(* Logix 5000 project; controller Final vendor 1 type 14 code 242 rev 32.11; software revision 32.00; part 2 of 2 *)
(* tags used below, declared in another part *)
   B_Pres1 : SensorType;   // Holds all values related to Brakes Pressure Sensor #1
   B_Pres2 : SensorType;   // Holds all values related to Brakes Pressure Sensor #2
   B_Pres3 : SensorType;   // Holds all values related to Brakes Pressure Sensor #3
   B_Pres4 : SensorType;   // Holds all values related to Brakes Pressure Sensor #4
   B_Pres5 : SensorType;   // Holds all values related to Brakes Pressure Sensor #5
   B_Pres6 : SensorType;   // Holds all values related to Brakes Pressure Sensor #6
   B_Pres7 : SensorType;   // Holds all values related to Brakes Pressure Sensor #7
   B_Pres8 : SensorType;   // Holds all values related to Brakes Pressure Sensor #8
   B_Pres9 : SensorType;   // Holds all values related to Brakes Pressure Sensor #9
   B_Tem0 : SensorType;   // Holds all values related to Brakes Temperature Sensor #0
   B_Tem1 : SensorType;   // Holds all values related to Brakes Temperature Sensor #1
   BATTERY_CHARGE : REAL;
   BATTERY_TEMP : REAL;
   BATTERY_VOLTAGE : REAL;
   BatteryA : REAL;
   BatteryB : REAL;
   BatteryC : REAL;
   bfr_SysSec : DINT;
   C_Las0 : SensorType;   // Holds all values related to Controls Laser Sensor #0
   C_Las1 : SensorType;   // Holds all values related to Controls Laser Sensor #1
   ConversionResistance : REAL;
   ConversionVoltage : REAL;
   count : DINT;
   Current_OoR : BOOL;
   InverseTemp : REAL;
   Limit1 : BOOL;
   Limit2 : BOOL;
   LogR : REAL;
   P_Pres0 : SensorType;   // Holds all values related to Pressure Pressure Sensor #0
   P_Pres1 : SensorType;   // Holds all values related to Pressure Pressure Sensor #1
   P_Pres2 : SensorType;   // Holds all values related to Pressure Pressure Sensor #2
   P_Pres3 : SensorType;
   P_Pres4 : SensorType;
   P_Tem1 : SensorType;   // Holds all values related to Pressure Temperature Sensor #1
   P_Tem2 : SensorType;
   P_Tem3 : SensorType;
   P_Tem4 : SensorType;
   S_B_Pres0 : SensorType;
   S_B_Pres1 : SensorType;
   S_B_Pres2 : SensorType;
   S_B_Pres3 : SensorType;
   S_B_Pres4 : SensorType;
   S_B_Pres5 : SensorType;
   S_B_Pres6 : SensorType;
   S_B_Pres7 : SensorType;
   S_B_Pres8 : SensorType;
   S_B_Pres9 : SensorType;
   S_B_Tem0 : SensorType;
   S_B_Tem1 : SensorType;
   S_BAT_FLAG : BOOL;
   S_BatteryC : DINT;
   S_BatteryT : REAL;
   S_BatteryV : REAL;
   S_BRAKE_FLAG : BOOL;
   S_Brake_Sub1 : DINT;
   S_Brake_Sub2 : DINT;
   S_COMMAND : DINT;
   S_COMN_FLAG : BOOL;
   S_COMN_STATE : BOOL;
   S_P_Pres1 : SensorType;
   S_P_Pres2 : SensorType;
   S_P_Pres3 : SensorType;
   S_P_Pres4 : SensorType;
   S_P_Tem1 : SensorType;
   S_P_Tem2 : SensorType;
   S_P_Tem3 : SensorType;
   S_P_Tem4 : SensorType;
   S_PROP_FLAG : BOOL;
   S_PROP_STATE : BOOL;
   S_STATE : DINT;
   S_Switch : AB:5000_DO4:O:0;
   S_SysFail : BOOL;
   sts_SysSec : DINT;
   Temperature_OoR : BOOL;
   tmr_HB : TIMER;   // TIMER Heartbeat
   Voltage_OoR : BOOL;
(* MainProgram, continued *)

ROUTINE Update_B_Pres1   (* structured text *)
   case B_Pres1.Count of
   	0: B_Pres1.PreviousValue0 := B_Pres1.CurrentValue;
   	1: B_Pres1.PreviousValue1 := B_Pres1.CurrentValue;
   	2: B_Pres1.PreviousValue2 := B_Pres1.CurrentValue;
   	3: B_Pres1.PreviousValue3 := B_Pres1.CurrentValue;
   	4: B_Pres1.PreviousValue4 := B_Pres1.CurrentValue;
   	5: B_Pres1.PreviousValue5 := B_Pres1.CurrentValue;
   	6: B_Pres1.PreviousValue6 := B_Pres1.CurrentValue;
   	7: B_Pres1.PreviousValue7 := B_Pres1.CurrentValue;
   	8: B_Pres1.PreviousValue8 := B_Pres1.CurrentValue;
   	9: B_Pres1.PreviousValue9 := B_Pres1.CurrentValue;
   end_case;
   B_Pres1.Count := B_Pres1.Count + 1;
   if B_Pres1.Count = 10 then
   	B_Pres1.Count := 0;
   	B_Pres1.MeanStart := 1;
   end_if;
   B_Pres1.CurrentValue := Local:1:I.Ch01.Data;
   if B_Pres1.MeanStart then
   	B_Pres1.Mean10 := (B_Pres1.PreviousValue0 + B_Pres1.PreviousValue1 + B_Pres1.PreviousValue2 + B_Pres1.PreviousValue3 + B_Pres1.PreviousValue4 + B_Pres1.PreviousValue5 + B_Pres1.PreviousValue6 + B_Pres1.PreviousValue7 + B_Pres1.PreviousValue8 + B_Pres1.PreviousValue9)/10;
   	B_Pres1.StanDev := SQRT(( (B_Pres1.PreviousValue0 - B_Pres1.Mean10)**2 + (B_Pres1.PreviousValue1 - B_Pres1.Mean10)**2 + (B_Pres1.PreviousValue2 - B_Pres1.Mean10)**2 + (B_Pres1.PreviousValue3 - B_Pres1.Mean10)**2 + (B_Pres1.PreviousValue4 - B_Pres1.Mean10)**2 + (B_Pres1.PreviousValue5 - B_Pres1.Mean10)**2 + (B_Pres1.PreviousValue6 - B_Pres1.Mean10)**2 + (B_Pres1.PreviousValue7 - B_Pres1.Mean10)**2 + (B_Pres1.PreviousValue8 - B_Pres1.Mean10)**2 + (B_Pres1.PreviousValue9 - B_Pres1.Mean10)**2)/10);
   end_if;
END_ROUTINE

ROUTINE Update_B_Pres2   (* structured text *)
   case B_Pres2.Count of
   	0: B_Pres2.PreviousValue0 := B_Pres2.CurrentValue;
   	1: B_Pres2.PreviousValue1 := B_Pres2.CurrentValue;
   	2: B_Pres2.PreviousValue2 := B_Pres2.CurrentValue;
   	3: B_Pres2.PreviousValue3 := B_Pres2.CurrentValue;
   	4: B_Pres2.PreviousValue4 := B_Pres2.CurrentValue;
   	5: B_Pres2.PreviousValue5 := B_Pres2.CurrentValue;
   	6: B_Pres2.PreviousValue6 := B_Pres2.CurrentValue;
   	7: B_Pres2.PreviousValue7 := B_Pres2.CurrentValue;
   	8: B_Pres2.PreviousValue8 := B_Pres2.CurrentValue;
   	9: B_Pres2.PreviousValue9 := B_Pres2.CurrentValue;
   end_case;
   B_Pres2.Count := B_Pres2.Count + 1;
   if B_Pres2.Count = 10 then
   	B_Pres2.Count := 0;
   	B_Pres2.MeanStart := 1;
   end_if;
   B_Pres2.CurrentValue := Local:1:I.Ch02.Data;
   if B_Pres2.MeanStart then
   	B_Pres2.Mean10 := (B_Pres2.PreviousValue0 + B_Pres2.PreviousValue1 + B_Pres2.PreviousValue2 + B_Pres2.PreviousValue3 + B_Pres2.PreviousValue4 + B_Pres2.PreviousValue5 + B_Pres2.PreviousValue6 + B_Pres2.PreviousValue7 + B_Pres2.PreviousValue8 + B_Pres2.PreviousValue9)/10;
   	B_Pres2.StanDev := SQRT(((B_Pres2.PreviousValue0 - B_Pres2.Mean10)**2 + (B_Pres2.PreviousValue1 - B_Pres2.Mean10)**2 + (B_Pres2.PreviousValue2 - B_Pres2.Mean10)**2 + (B_Pres2.PreviousValue3 - B_Pres2.Mean10)**2 + (B_Pres2.PreviousValue4 - B_Pres2.Mean10)**2 + (B_Pres2.PreviousValue5 - B_Pres2.Mean10)**2 + (B_Pres2.PreviousValue6 - B_Pres2.Mean10)**2 + (B_Pres2.PreviousValue7 - B_Pres2.Mean10)**2 + (B_Pres2.PreviousValue8 - B_Pres2.Mean10)**2 + (B_Pres2.PreviousValue9 - B_Pres2.Mean10)**2)/10);
   end_if;
END_ROUTINE

ROUTINE Update_B_Pres3   (* structured text *)
   case B_Pres3.Count of
   	0: B_Pres3.PreviousValue0 := B_Pres3.CurrentValue;
   	1: B_Pres3.PreviousValue1 := B_Pres3.CurrentValue;
   	2: B_Pres3.PreviousValue2 := B_Pres3.CurrentValue;
   	3: B_Pres3.PreviousValue3 := B_Pres3.CurrentValue;
   	4: B_Pres3.PreviousValue4 := B_Pres3.CurrentValue;
   	5: B_Pres3.PreviousValue5 := B_Pres3.CurrentValue;
   	6: B_Pres3.PreviousValue6 := B_Pres3.CurrentValue;
   	7: B_Pres3.PreviousValue7 := B_Pres3.CurrentValue;
   	8: B_Pres3.PreviousValue8 := B_Pres3.CurrentValue;
   	9: B_Pres3.PreviousValue9 := B_Pres3.CurrentValue;
   end_case;
   B_Pres3.Count := B_Pres3.Count + 1;
   if B_Pres3.Count = 10 then
   	B_Pres3.Count := 0;
   	B_Pres3.MeanStart := 1;
   end_if;
   B_Pres3.CurrentValue := Local:1:I.Ch03.Data;
   if B_Pres3.MeanStart then
   	B_Pres3.Mean10 := (B_Pres3.PreviousValue0 + B_Pres3.PreviousValue1 + B_Pres3.PreviousValue2 + B_Pres3.PreviousValue3 + B_Pres3.PreviousValue4 + B_Pres3.PreviousValue5 + B_Pres3.PreviousValue6 + B_Pres3.PreviousValue7 + B_Pres3.PreviousValue8 + B_Pres3.PreviousValue9)/10;
   	B_Pres3.StanDev := SQRT(((B_Pres3.PreviousValue0 - B_Pres3.Mean10)**2 + (B_Pres3.PreviousValue1 - B_Pres3.Mean10)**2 + (B_Pres3.PreviousValue2 - B_Pres3.Mean10)**2 + (B_Pres3.PreviousValue3 - B_Pres3.Mean10)**2 + (B_Pres3.PreviousValue4 - B_Pres3.Mean10)**2 + (B_Pres3.PreviousValue5 - B_Pres3.Mean10)**2 + (B_Pres3.PreviousValue6 - B_Pres3.Mean10)**2 + (B_Pres3.PreviousValue7 - B_Pres3.Mean10)**2 + (B_Pres3.PreviousValue8 - B_Pres3.Mean10)**2 + (B_Pres3.PreviousValue9 - B_Pres3.Mean10)**2)/10);
   end_if;
END_ROUTINE

ROUTINE Update_B_Pres4   (* structured text *)
   case B_Pres4.Count of
   	0: B_Pres4.PreviousValue0 := B_Pres4.CurrentValue;
   	1: B_Pres4.PreviousValue1 := B_Pres4.CurrentValue;
   	2: B_Pres4.PreviousValue2 := B_Pres4.CurrentValue;
   	3: B_Pres4.PreviousValue3 := B_Pres4.CurrentValue;
   	4: B_Pres4.PreviousValue4 := B_Pres4.CurrentValue;
   	5: B_Pres4.PreviousValue5 := B_Pres4.CurrentValue;
   	6: B_Pres4.PreviousValue6 := B_Pres4.CurrentValue;
   	7: B_Pres4.PreviousValue7 := B_Pres4.CurrentValue;
   	8: B_Pres4.PreviousValue8 := B_Pres4.CurrentValue;
   	9: B_Pres4.PreviousValue9 := B_Pres4.CurrentValue;
   end_case;
   B_Pres4.Count := B_Pres4.Count + 1;
   if B_Pres4.Count = 10 then
   	B_Pres4.Count := 0;
   	B_Pres4.MeanStart := 1;
   end_if;
   B_Pres4.CurrentValue := Local:1:I.Ch04.Data;
   if B_Pres4.MeanStart then
   	B_Pres4.Mean10 := (B_Pres4.PreviousValue0 + B_Pres4.PreviousValue1 + B_Pres4.PreviousValue2 + B_Pres4.PreviousValue3 + B_Pres4.PreviousValue4 + B_Pres4.PreviousValue5 + B_Pres4.PreviousValue6 + B_Pres4.PreviousValue7 + B_Pres4.PreviousValue8 + B_Pres4.PreviousValue9)/10;
   	B_Pres4.StanDev := SQRT(((B_Pres4.PreviousValue0 - B_Pres4.Mean10)**2 + (B_Pres4.PreviousValue1 - B_Pres4.Mean10)**2 + (B_Pres4.PreviousValue2 - B_Pres4.Mean10)**2 + (B_Pres4.PreviousValue3 - B_Pres4.Mean10)**2 + (B_Pres4.PreviousValue4 - B_Pres4.Mean10)**2 + (B_Pres4.PreviousValue5 - B_Pres4.Mean10)**2 + (B_Pres4.PreviousValue6 - B_Pres4.Mean10)**2 + (B_Pres4.PreviousValue7 - B_Pres4.Mean10)**2 + (B_Pres4.PreviousValue8 - B_Pres4.Mean10)**2 + (B_Pres4.PreviousValue9 - B_Pres4.Mean10)**2)/10);
   end_if;
END_ROUTINE

ROUTINE Update_B_Pres5   (* structured text *)
   case B_Pres5.Count of
   	0: B_Pres5.PreviousValue0 := B_Pres5.CurrentValue;
   	1: B_Pres5.PreviousValue1 := B_Pres5.CurrentValue;
   	2: B_Pres5.PreviousValue2 := B_Pres5.CurrentValue;
   	3: B_Pres5.PreviousValue3 := B_Pres5.CurrentValue;
   	4: B_Pres5.PreviousValue4 := B_Pres5.CurrentValue;
   	5: B_Pres5.PreviousValue5 := B_Pres5.CurrentValue;
   	6: B_Pres5.PreviousValue6 := B_Pres5.CurrentValue;
   	7: B_Pres5.PreviousValue7 := B_Pres5.CurrentValue;
   	8: B_Pres5.PreviousValue8 := B_Pres5.CurrentValue;
   	9: B_Pres5.PreviousValue9 := B_Pres5.CurrentValue;
   end_case;
   B_Pres5.Count := B_Pres5.Count + 1;
   if B_Pres5.Count = 10 then
   	B_Pres5.Count := 0;
   	B_Pres5.MeanStart := 1;
   end_if;
   B_Pres5.CurrentValue := Local:1:I.Ch05.Data;
   if B_Pres5.MeanStart then
   	B_Pres5.Mean10 := (B_Pres5.PreviousValue0 + B_Pres5.PreviousValue1 + B_Pres5.PreviousValue2 + B_Pres5.PreviousValue3 + B_Pres5.PreviousValue4 + B_Pres5.PreviousValue5 + B_Pres5.PreviousValue6 + B_Pres5.PreviousValue7 + B_Pres5.PreviousValue8 + B_Pres5.PreviousValue9)/10;
   	B_Pres5.StanDev := SQRT(((B_Pres5.PreviousValue0 - B_Pres5.Mean10)**2 + (B_Pres5.PreviousValue1 - B_Pres5.Mean10)**2 + (B_Pres5.PreviousValue2 - B_Pres5.Mean10)**2 + (B_Pres5.PreviousValue3 - B_Pres5.Mean10)**2 + (B_Pres5.PreviousValue4 - B_Pres5.Mean10)**2 + (B_Pres5.PreviousValue5 - B_Pres5.Mean10)**2 + (B_Pres5.PreviousValue6 - B_Pres5.Mean10)**2 + (B_Pres5.PreviousValue7 - B_Pres5.Mean10)**2 + (B_Pres5.PreviousValue8 - B_Pres5.Mean10)**2 + (B_Pres5.PreviousValue9 - B_Pres5.Mean10)**2)/10);
   end_if;
END_ROUTINE

ROUTINE Update_B_Pres6   (* structured text *)
   case B_Pres6.Count of
   	0: B_Pres6.PreviousValue0 := B_Pres6.CurrentValue;
   	1: B_Pres6.PreviousValue1 := B_Pres6.CurrentValue;
   	2: B_Pres6.PreviousValue2 := B_Pres6.CurrentValue;
   	3: B_Pres6.PreviousValue3 := B_Pres6.CurrentValue;
   	4: B_Pres6.PreviousValue4 := B_Pres6.CurrentValue;
   	5: B_Pres6.PreviousValue5 := B_Pres6.CurrentValue;
   	6: B_Pres6.PreviousValue6 := B_Pres6.CurrentValue;
   	7: B_Pres6.PreviousValue7 := B_Pres6.CurrentValue;
   	8: B_Pres6.PreviousValue8 := B_Pres6.CurrentValue;
   	9: B_Pres6.PreviousValue9 := B_Pres6.CurrentValue;
   end_case;
   B_Pres6.Count := B_Pres6.Count + 1;
   if B_Pres6.Count = 10 then
   	B_Pres6.Count := 0;
   	B_Pres6.MeanStart := 1;
   end_if;
   B_Pres6.CurrentValue := Local:1:I.Ch06.Data;
   if B_Pres6.MeanStart then
   	B_Pres6.Mean10 := (B_Pres6.PreviousValue0 + B_Pres6.PreviousValue1 + B_Pres6.PreviousValue2 + B_Pres6.PreviousValue3 + B_Pres6.PreviousValue4 + B_Pres6.PreviousValue5 + B_Pres6.PreviousValue6 + B_Pres6.PreviousValue7 + B_Pres6.PreviousValue8 + B_Pres6.PreviousValue9)/10;
   	B_Pres6.StanDev := SQRT(((B_Pres6.PreviousValue0 - B_Pres6.Mean10)**2 + (B_Pres6.PreviousValue1 - B_Pres6.Mean10)**2 + (B_Pres6.PreviousValue2 - B_Pres6.Mean10)**2 + (B_Pres6.PreviousValue3 - B_Pres6.Mean10)**2 + (B_Pres6.PreviousValue4 - B_Pres6.Mean10)**2 + (B_Pres6.PreviousValue5 - B_Pres6.Mean10)**2 + (B_Pres6.PreviousValue6 - B_Pres6.Mean10)**2 + (B_Pres6.PreviousValue7 - B_Pres6.Mean10)**2 + (B_Pres6.PreviousValue8 - B_Pres6.Mean10)**2 + (B_Pres6.PreviousValue9 - B_Pres6.Mean10)**2)/10);
   end_if;
END_ROUTINE

ROUTINE Update_B_Pres7   (* structured text *)
   case B_Pres7.Count of
   	0: B_Pres7.PreviousValue0 := B_Pres7.CurrentValue;
   	1: B_Pres7.PreviousValue1 := B_Pres7.CurrentValue;
   	2: B_Pres7.PreviousValue2 := B_Pres7.CurrentValue;
   	3: B_Pres7.PreviousValue3 := B_Pres7.CurrentValue;
   	4: B_Pres7.PreviousValue4 := B_Pres7.CurrentValue;
   	5: B_Pres7.PreviousValue5 := B_Pres7.CurrentValue;
   	6: B_Pres7.PreviousValue6 := B_Pres7.CurrentValue;
   	7: B_Pres7.PreviousValue7 := B_Pres7.CurrentValue;
   	8: B_Pres7.PreviousValue8 := B_Pres7.CurrentValue;
   	9: B_Pres7.PreviousValue9 := B_Pres7.CurrentValue;
   end_case;
   B_Pres7.Count := B_Pres7.Count + 1;
   if B_Pres7.Count = 10 then
   	B_Pres7.Count := 0;
   	B_Pres7.MeanStart := 1;
   end_if;
   B_Pres7.CurrentValue := Local:1:I.Ch07.Data;
   if B_Pres7.MeanStart then
   	B_Pres7.Mean10 := (B_Pres7.PreviousValue0 + B_Pres7.PreviousValue1 + B_Pres7.PreviousValue2 + B_Pres7.PreviousValue3 + B_Pres7.PreviousValue4 + B_Pres7.PreviousValue5 + B_Pres7.PreviousValue6 + B_Pres7.PreviousValue7 + B_Pres7.PreviousValue8 + B_Pres7.PreviousValue9)/10;
   	B_Pres7.StanDev := SQRT(((B_Pres7.PreviousValue0 - B_Pres7.Mean10)**2 + (B_Pres7.PreviousValue1 - B_Pres7.Mean10)**2 + (B_Pres7.PreviousValue2 - B_Pres7.Mean10)**2 + (B_Pres7.PreviousValue3 - B_Pres7.Mean10)**2 + (B_Pres7.PreviousValue4 - B_Pres7.Mean10)**2 + (B_Pres7.PreviousValue5 - B_Pres7.Mean10)**2 + (B_Pres7.PreviousValue6 - B_Pres7.Mean10)**2 + (B_Pres7.PreviousValue7 - B_Pres7.Mean10)**2 + (B_Pres7.PreviousValue8 - B_Pres7.Mean10)**2 + (B_Pres7.PreviousValue9 - B_Pres7.Mean10)**2)/10);
   end_if;
END_ROUTINE

ROUTINE Update_B_Pres8   (* structured text *)
   case B_Pres8.Count of
   	0: B_Pres8.PreviousValue0 := B_Pres8.CurrentValue;
   	1: B_Pres8.PreviousValue1 := B_Pres8.CurrentValue;
   	2: B_Pres8.PreviousValue2 := B_Pres8.CurrentValue;
   	3: B_Pres8.PreviousValue3 := B_Pres8.CurrentValue;
   	4: B_Pres8.PreviousValue4 := B_Pres8.CurrentValue;
   	5: B_Pres8.PreviousValue5 := B_Pres8.CurrentValue;
   	6: B_Pres8.PreviousValue6 := B_Pres8.CurrentValue;
   	7: B_Pres8.PreviousValue7 := B_Pres8.CurrentValue;
   	8: B_Pres8.PreviousValue8 := B_Pres8.CurrentValue;
   	9: B_Pres8.PreviousValue9 := B_Pres8.CurrentValue;
   end_case;
   B_Pres8.Count := B_Pres8.Count + 1;
   if B_Pres8.Count = 10 then
   	B_Pres8.Count := 0;
   	B_Pres8.MeanStart := 1;
   end_if;
   B_Pres8.CurrentValue := Local:2:I.Ch00.Data;
   if B_Pres8.MeanStart then
   	B_Pres8.Mean10 := (B_Pres8.PreviousValue0 + B_Pres8.PreviousValue1 + B_Pres8.PreviousValue2 + B_Pres8.PreviousValue3 + B_Pres8.PreviousValue4 + B_Pres8.PreviousValue5 + B_Pres8.PreviousValue6 + B_Pres8.PreviousValue7 + B_Pres8.PreviousValue8 + B_Pres8.PreviousValue9)/10;
   	B_Pres8.StanDev := SQRT(((B_Pres8.PreviousValue0 - B_Pres8.Mean10)**2 + (B_Pres8.PreviousValue1 - B_Pres8.Mean10)**2 + (B_Pres8.PreviousValue2 - B_Pres8.Mean10)**2 + (B_Pres8.PreviousValue3 - B_Pres8.Mean10)**2 + (B_Pres8.PreviousValue4 - B_Pres8.Mean10)**2 + (B_Pres8.PreviousValue5 - B_Pres8.Mean10)**2 + (B_Pres8.PreviousValue6 - B_Pres8.Mean10)**2 + (B_Pres8.PreviousValue7 - B_Pres8.Mean10)**2 + (B_Pres8.PreviousValue8 - B_Pres8.Mean10)**2 + (B_Pres8.PreviousValue9 - B_Pres8.Mean10)**2)/10);
   end_if;
END_ROUTINE

ROUTINE Update_B_Pres9   (* structured text *)
   case B_Pres9.Count of
   	0: B_Pres9.PreviousValue0 := B_Pres9.CurrentValue;
   	1: B_Pres9.PreviousValue1 := B_Pres9.CurrentValue;
   	2: B_Pres9.PreviousValue2 := B_Pres9.CurrentValue;
   	3: B_Pres9.PreviousValue3 := B_Pres9.CurrentValue;
   	4: B_Pres9.PreviousValue4 := B_Pres9.CurrentValue;
   	5: B_Pres9.PreviousValue5 := B_Pres9.CurrentValue;
   	6: B_Pres9.PreviousValue6 := B_Pres9.CurrentValue;
   	7: B_Pres9.PreviousValue7 := B_Pres9.CurrentValue;
   	8: B_Pres9.PreviousValue8 := B_Pres9.CurrentValue;
   	9: B_Pres9.PreviousValue9 := B_Pres9.CurrentValue;
   end_case;
   B_Pres9.Count := B_Pres9.Count + 1;
   if B_Pres9.Count = 10 then
   	B_Pres9.Count := 0;
   	B_Pres9.MeanStart := 1;
   end_if;
   B_Pres9.CurrentValue := Local:2:I.Ch01.Data;
   if B_Pres9.MeanStart then
   	B_Pres9.Mean10 := (B_Pres9.PreviousValue0 + B_Pres9.PreviousValue1 + B_Pres9.PreviousValue2 + B_Pres9.PreviousValue3 + B_Pres9.PreviousValue4 + B_Pres9.PreviousValue5 + B_Pres9.PreviousValue6 + B_Pres9.PreviousValue7 + B_Pres9.PreviousValue8 + B_Pres9.PreviousValue9)/10;
   	B_Pres9.StanDev := SQRT(((B_Pres9.PreviousValue0 - B_Pres9.Mean10)**2 + (B_Pres9.PreviousValue1 - B_Pres9.Mean10)**2 + (B_Pres9.PreviousValue2 - B_Pres9.Mean10)**2 + (B_Pres9.PreviousValue3 - B_Pres9.Mean10)**2 + (B_Pres9.PreviousValue4 - B_Pres9.Mean10)**2 + (B_Pres9.PreviousValue5 - B_Pres9.Mean10)**2 + (B_Pres9.PreviousValue6 - B_Pres9.Mean10)**2 + (B_Pres9.PreviousValue7 - B_Pres9.Mean10)**2 + (B_Pres9.PreviousValue8 - B_Pres9.Mean10)**2 + (B_Pres9.PreviousValue9 - B_Pres9.Mean10)**2)/10);
   end_if;
END_ROUTINE

ROUTINE Update_B_Tem0   (* structured text *)
   case B_Tem0.Count of
   	0: B_Tem0.PreviousValue0 := B_Tem0.CurrentValue;
   	1: B_Tem0.PreviousValue1 := B_Tem0.CurrentValue;
   	2: B_Tem0.PreviousValue2 := B_Tem0.CurrentValue;
   	3: B_Tem0.PreviousValue3 := B_Tem0.CurrentValue;
   	4: B_Tem0.PreviousValue4 := B_Tem0.CurrentValue;
   	5: B_Tem0.PreviousValue5 := B_Tem0.CurrentValue;
   	6: B_Tem0.PreviousValue6 := B_Tem0.CurrentValue;
   	7: B_Tem0.PreviousValue7 := B_Tem0.CurrentValue;
   	8: B_Tem0.PreviousValue8 := B_Tem0.CurrentValue;
   	9: B_Tem0.PreviousValue9 := B_Tem0.CurrentValue;
   end_case;
   B_Tem0.Count := B_Tem0.Count + 1;
   if B_Tem0.Count = 10 then
   	B_Tem0.Count := 0;
   	B_Tem0.MeanStart := 1;
   end_if;
   B_Tem0.CurrentValue := Local:2:I.Ch02.Data;
   if B_Tem0.MeanStart then
   	B_Tem0.Mean10 := (B_Tem0.PreviousValue0 + B_Tem0.PreviousValue1 + B_Tem0.PreviousValue2 + B_Tem0.PreviousValue3 + B_Tem0.PreviousValue4 + B_Tem0.PreviousValue5 + B_Tem0.PreviousValue6 + B_Tem0.PreviousValue7 + B_Tem0.PreviousValue8 + B_Tem0.PreviousValue9)/10;
   	B_Tem0.StanDev := SQRT(((B_Tem0.PreviousValue0 - B_Tem0.Mean10)**2 + (B_Tem0.PreviousValue1 - B_Tem0.Mean10)**2 + (B_Tem0.PreviousValue2 - B_Tem0.Mean10)**2 + (B_Tem0.PreviousValue3 - B_Tem0.Mean10)**2 + (B_Tem0.PreviousValue4 - B_Tem0.Mean10)**2 + (B_Tem0.PreviousValue5 - B_Tem0.Mean10)**2 + (B_Tem0.PreviousValue6 - B_Tem0.Mean10)**2 + (B_Tem0.PreviousValue7 - B_Tem0.Mean10)**2 + (B_Tem0.PreviousValue8 - B_Tem0.Mean10)**2 + (B_Tem0.PreviousValue9 - B_Tem0.Mean10)**2)/10);
   end_if;
END_ROUTINE

ROUTINE Update_B_Tem1   (* structured text *)
   case B_Tem1.Count of
   	0: B_Tem1.PreviousValue0 := B_Tem1.CurrentValue;
   	1: B_Tem1.PreviousValue1 := B_Tem1.CurrentValue;
   	2: B_Tem1.PreviousValue2 := B_Tem1.CurrentValue;
   	3: B_Tem1.PreviousValue3 := B_Tem1.CurrentValue;
   	4: B_Tem1.PreviousValue4 := B_Tem1.CurrentValue;
   	5: B_Tem1.PreviousValue5 := B_Tem1.CurrentValue;
   	6: B_Tem1.PreviousValue6 := B_Tem1.CurrentValue;
   	7: B_Tem1.PreviousValue7 := B_Tem1.CurrentValue;
   	8: B_Tem1.PreviousValue8 := B_Tem1.CurrentValue;
   	9: B_Tem1.PreviousValue9 := B_Tem1.CurrentValue;
   end_case;
   B_Tem1.Count := B_Tem1.Count + 1;
   if B_Tem1.Count = 10 then
   	B_Tem1.Count := 0;
   	B_Tem1.MeanStart := 1;
   end_if;
   B_Tem1.CurrentValue := Local:2:I.Ch03.Data;
   if B_Tem1.MeanStart then
   	B_Tem1.Mean10 := (B_Tem1.PreviousValue0 + B_Tem1.PreviousValue1 + B_Tem1.PreviousValue2 + B_Tem1.PreviousValue3 + B_Tem1.PreviousValue4 + B_Tem1.PreviousValue5 + B_Tem1.PreviousValue6 + B_Tem1.PreviousValue7 + B_Tem1.PreviousValue8 + B_Tem1.PreviousValue9)/10;
   	B_Tem1.StanDev := SQRT(((B_Tem1.PreviousValue0 - B_Tem1.Mean10)**2 + (B_Tem1.PreviousValue1 - B_Tem1.Mean10)**2 + (B_Tem1.PreviousValue2 - B_Tem1.Mean10)**2 + (B_Tem1.PreviousValue3 - B_Tem1.Mean10)**2 + (B_Tem1.PreviousValue4 - B_Tem1.Mean10)**2 + (B_Tem1.PreviousValue5 - B_Tem1.Mean10)**2 + (B_Tem1.PreviousValue6 - B_Tem1.Mean10)**2 + (B_Tem1.PreviousValue7 - B_Tem1.Mean10)**2 + (B_Tem1.PreviousValue8 - B_Tem1.Mean10)**2 + (B_Tem1.PreviousValue9 - B_Tem1.Mean10)**2)/10);
   end_if;
END_ROUTINE

ROUTINE Update_Battery_Amp   (* structured text *)
   
END_ROUTINE

ROUTINE Update_Battery_Temp   (* structured text *)
   ConversionVoltage := Local:2:I.Ch06.Data;
   ConversionResistance := 12650 * (5 - ConversionVoltage) / ConversionVoltage;
   BatteryA := 0.00112924;//-0.0005697945479763659;//25.633751435943907;//
   BatteryB := 0.000234108;//0.0005112936453520823;//-20.64469507056110;//
   BatteryC := 0.000000087755;//-0.0000008923754330128293;//-0.338811414517226;//
   LogR := LN(ConversionResistance);
   InverseTemp := BatteryA + BatteryB * LogR + BatteryC * (LogR ** 3);
   BATTERY_TEMP := 1 / InverseTemp ;//- 45;
END_ROUTINE

ROUTINE Update_Battery_Volt   (* structured text *)
   BATTERY_VOLTAGE := Local:2:I.Ch05.Data;
   BATTERY_CHARGE := (BATTERY_VOLTAGE - 23) * 100 / 6;
END_ROUTINE

ROUTINE Update_C_Las0   (* structured text *)
   case C_Las0.Count of
   	0: C_Las0.PreviousValue0 := C_Las0.CurrentValue;
   	1: C_Las0.PreviousValue1 := C_Las0.CurrentValue;
   	2: C_Las0.PreviousValue2 := C_Las0.CurrentValue;
   	3: C_Las0.PreviousValue3 := C_Las0.CurrentValue;
   	4: C_Las0.PreviousValue4 := C_Las0.CurrentValue;
   	5: C_Las0.PreviousValue5 := C_Las0.CurrentValue;
   	6: C_Las0.PreviousValue6 := C_Las0.CurrentValue;
   	7: C_Las0.PreviousValue7 := C_Las0.CurrentValue;
   	8: C_Las0.PreviousValue8 := C_Las0.CurrentValue;
   	9: C_Las0.PreviousValue9 := C_Las0.CurrentValue;
   end_case;
   C_Las0.Count := C_Las0.Count + 1;
   if C_Las0.Count = 10 then
   	C_Las0.Count := 0;
   	C_Las0.MeanStart := 1;
   end_if;
   C_Las0.CurrentValue := Local:7:I.Counter00.Count;
   if C_Las0.MeanStart then
   	C_Las0.Mean10 := (C_Las0.PreviousValue0 + C_Las0.PreviousValue1 + C_Las0.PreviousValue2 + C_Las0.PreviousValue3 + C_Las0.PreviousValue4 + C_Las0.PreviousValue5 + C_Las0.PreviousValue6 + C_Las0.PreviousValue7 + C_Las0.PreviousValue8 + C_Las0.PreviousValue9)/10;
   	C_Las0.StanDev := SQRT(((C_Las0.PreviousValue0 - C_Las0.Mean10)**2 + (C_Las0.PreviousValue1 - C_Las0.Mean10)**2 + (C_Las0.PreviousValue2 - C_Las0.Mean10)**2 + (C_Las0.PreviousValue3 - C_Las0.Mean10)**2 + (C_Las0.PreviousValue4 - C_Las0.Mean10)**2 + (C_Las0.PreviousValue5 - C_Las0.Mean10)**2 + (C_Las0.PreviousValue6 - C_Las0.Mean10)**2 + (C_Las0.PreviousValue7 - C_Las0.Mean10)**2 + (C_Las0.PreviousValue8 - C_Las0.Mean10)**2 + (C_Las0.PreviousValue9 - C_Las0.Mean10)**2)/10);
   end_if;
END_ROUTINE

ROUTINE Update_C_Las1   (* structured text *)
   case C_Las1.Count of
   	0: C_Las1.PreviousValue0 := C_Las1.CurrentValue;
   	1: C_Las1.PreviousValue1 := C_Las1.CurrentValue;
   	2: C_Las1.PreviousValue2 := C_Las1.CurrentValue;
   	3: C_Las1.PreviousValue3 := C_Las1.CurrentValue;
   	4: C_Las1.PreviousValue4 := C_Las1.CurrentValue;
   	5: C_Las1.PreviousValue5 := C_Las1.CurrentValue;
   	6: C_Las1.PreviousValue6 := C_Las1.CurrentValue;
   	7: C_Las1.PreviousValue7 := C_Las1.CurrentValue;
   	8: C_Las1.PreviousValue8 := C_Las1.CurrentValue;
   	9: C_Las1.PreviousValue9 := C_Las1.CurrentValue;
   end_case;
   C_Las1.Count := C_Las1.Count + 1;
   if C_Las1.Count = 10 then
   	C_Las1.Count := 0;
   	C_Las1.MeanStart := 1;
   end_if;
   C_Las1.CurrentValue := Local:7:I.Counter01.Count;
   if C_Las1.MeanStart then
   	C_Las1.Mean10 := (C_Las1.PreviousValue0 + C_Las1.PreviousValue1 + C_Las1.PreviousValue2 + C_Las1.PreviousValue3 + C_Las1.PreviousValue4 + C_Las1.PreviousValue5 + C_Las1.PreviousValue6 + C_Las1.PreviousValue7 + C_Las1.PreviousValue8 + C_Las1.PreviousValue9)/10;
   	C_Las1.StanDev := SQRT(((C_Las1.PreviousValue0 - C_Las1.Mean10)**2 + (C_Las1.PreviousValue1 - C_Las1.Mean10)**2 + (C_Las1.PreviousValue2 - C_Las1.Mean10)**2 + (C_Las1.PreviousValue3 - C_Las1.Mean10)**2 + (C_Las1.PreviousValue4 - C_Las1.Mean10)**2 + (C_Las1.PreviousValue5 - C_Las1.Mean10)**2 + (C_Las1.PreviousValue6 - C_Las1.Mean10)**2 + (C_Las1.PreviousValue7 - C_Las1.Mean10)**2 + (C_Las1.PreviousValue8 - C_Las1.Mean10)**2 + (C_Las1.PreviousValue9 - C_Las1.Mean10)**2)/10);
   end_if;
END_ROUTINE

ROUTINE Update_Limit1   (* structured text *)
   Limit1 := Local:6:I.Pt00.Data;
END_ROUTINE

ROUTINE Update_Limit2   (* structured text *)
   Limit2 := Local:6:I.Pt01.Data;
END_ROUTINE

ROUTINE Update_P_Pres0   (* structured text *)
   case P_Pres0.Count of
   	0: P_Pres0.PreviousValue0 := P_Pres0.CurrentValue;
   	1: P_Pres0.PreviousValue1 := P_Pres0.CurrentValue;
   	2: P_Pres0.PreviousValue2 := P_Pres0.CurrentValue;
   	3: P_Pres0.PreviousValue3 := P_Pres0.CurrentValue;
   	4: P_Pres0.PreviousValue4 := P_Pres0.CurrentValue;
   	5: P_Pres0.PreviousValue5 := P_Pres0.CurrentValue;
   	6: P_Pres0.PreviousValue6 := P_Pres0.CurrentValue;
   	7: P_Pres0.PreviousValue7 := P_Pres0.CurrentValue;
   	8: P_Pres0.PreviousValue8 := P_Pres0.CurrentValue;
   	9: P_Pres0.PreviousValue9 := P_Pres0.CurrentValue;
   end_case;
   P_Pres0.Count := P_Pres0.Count + 1;
   if P_Pres0.Count = 10 then
   	P_Pres0.Count := 0;
   	P_Pres0.MeanStart := 1;
   end_if;
   P_Pres0.CurrentValue := Local:2:I.Ch04.Data;
   if P_Pres0.MeanStart then
   	P_Pres0.Mean10 := (P_Pres0.PreviousValue0 + P_Pres0.PreviousValue1 + P_Pres0.PreviousValue2 + P_Pres0.PreviousValue3 + P_Pres0.PreviousValue4 + P_Pres0.PreviousValue5 + P_Pres0.PreviousValue6 + P_Pres0.PreviousValue7 + P_Pres0.PreviousValue8 + P_Pres0.PreviousValue9)/10;
   	P_Pres0.StanDev := SQRT(((P_Pres0.PreviousValue0 - P_Pres0.Mean10)**2 + (P_Pres0.PreviousValue1 - P_Pres0.Mean10)**2 + (P_Pres0.PreviousValue2 - P_Pres0.Mean10)**2 + (P_Pres0.PreviousValue3 - P_Pres0.Mean10)**2 + (P_Pres0.PreviousValue4 - P_Pres0.Mean10)**2 + (P_Pres0.PreviousValue5 - P_Pres0.Mean10)**2 + (P_Pres0.PreviousValue6 - P_Pres0.Mean10)**2 + (P_Pres0.PreviousValue7 - P_Pres0.Mean10)**2 + (P_Pres0.PreviousValue8 - P_Pres0.Mean10)**2 + (P_Pres0.PreviousValue9 - P_Pres0.Mean10)**2)/10);
   end_if;
END_ROUTINE

ROUTINE Update_P_Pres1   (* structured text *)
   case P_Pres1.Count of
   	0: P_Pres1.PreviousValue0 := P_Pres1.CurrentValue;
   	1: P_Pres1.PreviousValue1 := P_Pres1.CurrentValue;
   	2: P_Pres1.PreviousValue2 := P_Pres1.CurrentValue;
   	3: P_Pres1.PreviousValue3 := P_Pres1.CurrentValue;
   	4: P_Pres1.PreviousValue4 := P_Pres1.CurrentValue;
   	5: P_Pres1.PreviousValue5 := P_Pres1.CurrentValue;
   	6: P_Pres1.PreviousValue6 := P_Pres1.CurrentValue;
   	7: P_Pres1.PreviousValue7 := P_Pres1.CurrentValue;
   	8: P_Pres1.PreviousValue8 := P_Pres1.CurrentValue;
   	9: P_Pres1.PreviousValue9 := P_Pres1.CurrentValue;
   end_case;
   P_Pres1.Count := P_Pres1.Count + 1;
   if P_Pres1.Count = 10 then
   	P_Pres1.Count := 0;
   	P_Pres0.MeanStart := 1;
   end_if;
   P_Pres1.CurrentValue := Local:3:I.Ch00.Data;
   if P_Pres1.MeanStart then
   	P_Pres1.Mean10 := (P_Pres1.PreviousValue0 + P_Pres1.PreviousValue1 + P_Pres1.PreviousValue2 + P_Pres1.PreviousValue3 + P_Pres1.PreviousValue4 + P_Pres1.PreviousValue5 + P_Pres1.PreviousValue6 + P_Pres1.PreviousValue7 + P_Pres1.PreviousValue8 + P_Pres1.PreviousValue9)/10;
   	P_Pres1.StanDev := SQRT(((P_Pres1.PreviousValue0 - P_Pres1.Mean10)**2 + (P_Pres1.PreviousValue1 - P_Pres1.Mean10)**2 + (P_Pres1.PreviousValue2 - P_Pres1.Mean10)**2 + (P_Pres1.PreviousValue3 - P_Pres1.Mean10)**2 + (P_Pres1.PreviousValue4 - P_Pres1.Mean10)**2 + (P_Pres1.PreviousValue5 - P_Pres1.Mean10)**2 + (P_Pres1.PreviousValue6 - P_Pres1.Mean10)**2 + (P_Pres1.PreviousValue7 - P_Pres1.Mean10)**2 + (P_Pres1.PreviousValue8 - P_Pres1.Mean10)**2 + (P_Pres1.PreviousValue9 - P_Pres1.Mean10)**2)/10);
   end_if;
END_ROUTINE

ROUTINE Update_P_Pres2   (* structured text *)
   case P_Pres2.Count of
   	0: P_Pres2.PreviousValue0 := P_Pres2.CurrentValue;
   	1: P_Pres2.PreviousValue1 := P_Pres2.CurrentValue;
   	2: P_Pres2.PreviousValue2 := P_Pres2.CurrentValue;
   	3: P_Pres2.PreviousValue3 := P_Pres2.CurrentValue;
   	4: P_Pres2.PreviousValue4 := P_Pres2.CurrentValue;
   	5: P_Pres2.PreviousValue5 := P_Pres2.CurrentValue;
   	6: P_Pres2.PreviousValue6 := P_Pres2.CurrentValue;
   	7: P_Pres2.PreviousValue7 := P_Pres2.CurrentValue;
   	8: P_Pres2.PreviousValue8 := P_Pres2.CurrentValue;
   	9: P_Pres2.PreviousValue9 := P_Pres2.CurrentValue;
   end_case;
   P_Pres2.Count := P_Pres2.Count + 1;
   if P_Pres2.Count = 10 then
   	P_Pres2.Count := 0;
   	P_Pres2.MeanStart := 1;
   end_if;
   P_Pres2.CurrentValue := Local:3:I.Ch01.Data;
   if P_Pres2.MeanStart then
   	P_Pres2.Mean10 := (P_Pres2.PreviousValue0 + P_Pres2.PreviousValue1 + P_Pres2.PreviousValue2 + P_Pres2.PreviousValue3 + P_Pres2.PreviousValue4 + P_Pres2.PreviousValue5 + P_Pres2.PreviousValue6 + P_Pres2.PreviousValue7 + P_Pres2.PreviousValue8 + P_Pres2.PreviousValue9)/10;
   	P_Pres2.StanDev := SQRT(((P_Pres2.PreviousValue0 - P_Pres2.Mean10)**2 + (P_Pres2.PreviousValue1 - P_Pres2.Mean10)**2 + (P_Pres2.PreviousValue2 - P_Pres2.Mean10)**2 + (P_Pres2.PreviousValue3 - P_Pres2.Mean10)**2 + (P_Pres2.PreviousValue4 - P_Pres2.Mean10)**2 + (P_Pres2.PreviousValue5 - P_Pres2.Mean10)**2 + (P_Pres2.PreviousValue6 - P_Pres2.Mean10)**2 + (P_Pres2.PreviousValue7 - P_Pres2.Mean10)**2 + (P_Pres2.PreviousValue8 - P_Pres2.Mean10)**2 + (P_Pres2.PreviousValue9 - P_Pres2.Mean10)**2)/10);
   end_if;
END_ROUTINE

ROUTINE Update_P_Pres3   (* structured text *)
   case P_Pres3.Count of
   	0: P_Pres3.PreviousValue0 := P_Pres3.CurrentValue;
   	1: P_Pres3.PreviousValue1 := P_Pres3.CurrentValue;
   	2: P_Pres3.PreviousValue2 := P_Pres3.CurrentValue;
   	3: P_Pres3.PreviousValue3 := P_Pres3.CurrentValue;
   	4: P_Pres3.PreviousValue4 := P_Pres3.CurrentValue;
   	5: P_Pres3.PreviousValue5 := P_Pres3.CurrentValue;
   	6: P_Pres3.PreviousValue6 := P_Pres3.CurrentValue;
   	7: P_Pres3.PreviousValue7 := P_Pres3.CurrentValue;
   	8: P_Pres3.PreviousValue8 := P_Pres3.CurrentValue;
   	9: P_Pres3.PreviousValue9 := P_Pres3.CurrentValue;
   end_case;
   P_Pres3.Count := P_Pres3.Count + 1;
   if P_Pres3.Count = 10 then
   	P_Pres3.Count := 0;
   	P_Pres3.MeanStart := 1;
   end_if;
   P_Pres3.CurrentValue := Local:3:I.Ch02.Data;
   if P_Pres3.MeanStart then
   	P_Pres3.Mean10 := (P_Pres3.PreviousValue0 + P_Pres3.PreviousValue1 + P_Pres3.PreviousValue2 + P_Pres3.PreviousValue3 + P_Pres3.PreviousValue4 + P_Pres3.PreviousValue5 + P_Pres3.PreviousValue6 + P_Pres3.PreviousValue7 + P_Pres3.PreviousValue8 + P_Pres3.PreviousValue9)/10;
   	P_Pres3.StanDev := SQRT(((P_Pres3.PreviousValue0 - P_Pres3.Mean10)**2 + (P_Pres3.PreviousValue1 - P_Pres3.Mean10)**2 + (P_Pres3.PreviousValue2 - P_Pres3.Mean10)**2 + (P_Pres3.PreviousValue3 - P_Pres3.Mean10)**2 + (P_Pres3.PreviousValue4 - P_Pres3.Mean10)**2 + (P_Pres3.PreviousValue5 - P_Pres3.Mean10)**2 + (P_Pres3.PreviousValue6 - P_Pres3.Mean10)**2 + (P_Pres3.PreviousValue7 - P_Pres3.Mean10)**2 + (P_Pres3.PreviousValue8 - P_Pres3.Mean10)**2 + (P_Pres3.PreviousValue9 - P_Pres3.Mean10)**2)/10);
   end_if;
END_ROUTINE

ROUTINE Update_P_Pres4   (* structured text *)
   case P_Pres4.Count of
   	0: P_Pres4.PreviousValue0 := P_Pres4.CurrentValue;
   	1: P_Pres4.PreviousValue1 := P_Pres4.CurrentValue;
   	2: P_Pres4.PreviousValue2 := P_Pres4.CurrentValue;
   	3: P_Pres4.PreviousValue3 := P_Pres4.CurrentValue;
   	4: P_Pres4.PreviousValue4 := P_Pres4.CurrentValue;
   	5: P_Pres4.PreviousValue5 := P_Pres4.CurrentValue;
   	6: P_Pres4.PreviousValue6 := P_Pres4.CurrentValue;
   	7: P_Pres4.PreviousValue7 := P_Pres4.CurrentValue;
   	8: P_Pres4.PreviousValue8 := P_Pres4.CurrentValue;
   	9: P_Pres4.PreviousValue9 := P_Pres4.CurrentValue;
   end_case;
   P_Pres4.Count := P_Pres4.Count + 1;
   if P_Pres4.Count = 10 then
   	P_Pres4.Count := 0;
   	P_Pres4.MeanStart := 1;
   end_if;
   P_Pres4.CurrentValue := Local:3:I.Ch03.Data;
   if P_Pres4.MeanStart then
   	P_Pres4.Mean10 := (P_Pres4.PreviousValue0 + P_Pres4.PreviousValue1 + P_Pres4.PreviousValue2 + P_Pres4.PreviousValue3 + P_Pres4.PreviousValue4 + P_Pres4.PreviousValue5 + P_Pres4.PreviousValue6 + P_Pres4.PreviousValue7 + P_Pres4.PreviousValue8 + P_Pres4.PreviousValue9)/10;
   	P_Pres4.StanDev := SQRT(((P_Pres4.PreviousValue0 - P_Pres4.Mean10)**2 + (P_Pres4.PreviousValue1 - P_Pres4.Mean10)**2 + (P_Pres4.PreviousValue2 - P_Pres4.Mean10)**2 + (P_Pres4.PreviousValue3 - P_Pres4.Mean10)**2 + (P_Pres4.PreviousValue4 - P_Pres4.Mean10)**2 + (P_Pres4.PreviousValue5 - P_Pres4.Mean10)**2 + (P_Pres4.PreviousValue6 - P_Pres4.Mean10)**2 + (P_Pres4.PreviousValue7 - P_Pres4.Mean10)**2 + (P_Pres4.PreviousValue8 - P_Pres4.Mean10)**2 + (P_Pres4.PreviousValue9 - P_Pres4.Mean10)**2)/10);
   end_if;
END_ROUTINE

ROUTINE Update_P_Tem1   (* structured text *)
   case P_Tem1.Count of
   	0: P_Tem1.PreviousValue0 := P_Tem1.CurrentValue;
   	1: P_Tem1.PreviousValue1 := P_Tem1.CurrentValue;
   	2: P_Tem1.PreviousValue2 := P_Tem1.CurrentValue;
   	3: P_Tem1.PreviousValue3 := P_Tem1.CurrentValue;
   	4: P_Tem1.PreviousValue4 := P_Tem1.CurrentValue;
   	5: P_Tem1.PreviousValue5 := P_Tem1.CurrentValue;
   	6: P_Tem1.PreviousValue6 := P_Tem1.CurrentValue;
   	7: P_Tem1.PreviousValue7 := P_Tem1.CurrentValue;
   	8: P_Tem1.PreviousValue8 := P_Tem1.CurrentValue;
   	9: P_Tem1.PreviousValue9 := P_Tem1.CurrentValue;
   end_case;
   P_Tem1.Count := P_Tem1.Count + 1;
   if P_Tem1.Count = 10 then
   	P_Tem1.Count := 0;
   	P_Tem1.MeanStart := 1;
   end_if;
   P_Tem1.CurrentValue := Local:3:I.Ch04.Data;
   if P_Tem1.MeanStart then
   	P_Tem1.Mean10 := (P_Tem1.PreviousValue0 + P_Tem1.PreviousValue1 + P_Tem1.PreviousValue2 + P_Tem1.PreviousValue3 + P_Tem1.PreviousValue4 + P_Tem1.PreviousValue5 + P_Tem1.PreviousValue6 + P_Tem1.PreviousValue7 + P_Tem1.PreviousValue8 + P_Tem1.PreviousValue9)/10;
   	P_Tem1.StanDev := SQRT(((P_Tem1.PreviousValue0 - P_Tem1.Mean10)**2 + (P_Tem1.PreviousValue1 - P_Tem1.Mean10)**2 + (P_Tem1.PreviousValue2 - P_Tem1.Mean10)**2 + (P_Tem1.PreviousValue3 - P_Tem1.Mean10)**2 + (P_Tem1.PreviousValue4 - P_Tem1.Mean10)**2 + (P_Tem1.PreviousValue5 - P_Tem1.Mean10)**2 + (P_Tem1.PreviousValue6 - P_Tem1.Mean10)**2 + (P_Tem1.PreviousValue7 - P_Tem1.Mean10)**2 + (P_Tem1.PreviousValue8 - P_Tem1.Mean10)**2 + (P_Tem1.PreviousValue9 - P_Tem1.Mean10)**2)/10);
   end_if;
END_ROUTINE

ROUTINE Update_P_Tem2   (* structured text *)
   case P_Tem2.Count of
   	0: P_Tem2.PreviousValue0 := P_Tem2.CurrentValue;
   	1: P_Tem2.PreviousValue1 := P_Tem2.CurrentValue;
   	2: P_Tem2.PreviousValue2 := P_Tem2.CurrentValue;
   	3: P_Tem2.PreviousValue3 := P_Tem2.CurrentValue;
   	4: P_Tem2.PreviousValue4 := P_Tem2.CurrentValue;
   	5: P_Tem2.PreviousValue5 := P_Tem2.CurrentValue;
   	6: P_Tem2.PreviousValue6 := P_Tem2.CurrentValue;
   	7: P_Tem2.PreviousValue7 := P_Tem2.CurrentValue;
   	8: P_Tem2.PreviousValue8 := P_Tem2.CurrentValue;
   	9: P_Tem2.PreviousValue9 := P_Tem2.CurrentValue;
   end_case;
   P_Tem2.Count := P_Tem2.Count + 1;
   if P_Tem2.Count = 10 then
   	P_Tem2.Count := 0;
   	P_Tem2.MeanStart := 1;
   end_if;
   P_Tem2.CurrentValue := Local:3:I.Ch05.Data;
   if P_Tem2.MeanStart then
   	P_Tem2.Mean10 := (P_Tem2.PreviousValue0 + P_Tem2.PreviousValue1 + P_Tem2.PreviousValue2 + P_Tem2.PreviousValue3 + P_Tem2.PreviousValue4 + P_Tem2.PreviousValue5 + P_Tem2.PreviousValue6 + P_Tem2.PreviousValue7 + P_Tem2.PreviousValue8 + P_Tem2.PreviousValue9)/10;
   	P_Tem2.StanDev := SQRT(((P_Tem2.PreviousValue0 - P_Tem2.Mean10)**2 + (P_Tem2.PreviousValue1 - P_Tem2.Mean10)**2 + (P_Tem2.PreviousValue2 - P_Tem2.Mean10)**2 + (P_Tem2.PreviousValue3 - P_Tem2.Mean10)**2 + (P_Tem2.PreviousValue4 - P_Tem2.Mean10)**2 + (P_Tem2.PreviousValue5 - P_Tem2.Mean10)**2 + (P_Tem2.PreviousValue6 - P_Tem2.Mean10)**2 + (P_Tem2.PreviousValue7 - P_Tem2.Mean10)**2 + (P_Tem2.PreviousValue8 - P_Tem2.Mean10)**2 + (P_Tem2.PreviousValue9 - P_Tem2.Mean10)**2)/10);
   end_if;
END_ROUTINE

ROUTINE Update_P_Tem3   (* structured text *)
   case P_Tem3.Count of
   	0: P_Tem3.PreviousValue0 := P_Tem3.CurrentValue;
   	1: P_Tem3.PreviousValue1 := P_Tem3.CurrentValue;
   	2: P_Tem3.PreviousValue2 := P_Tem3.CurrentValue;
   	3: P_Tem3.PreviousValue3 := P_Tem3.CurrentValue;
   	4: P_Tem3.PreviousValue4 := P_Tem3.CurrentValue;
   	5: P_Tem3.PreviousValue5 := P_Tem3.CurrentValue;
   	6: P_Tem3.PreviousValue6 := P_Tem3.CurrentValue;
   	7: P_Tem3.PreviousValue7 := P_Tem3.CurrentValue;
   	8: P_Tem3.PreviousValue8 := P_Tem3.CurrentValue;
   	9: P_Tem3.PreviousValue9 := P_Tem3.CurrentValue;
   end_case;
   P_Tem3.Count := P_Tem3.Count + 1;
   if P_Tem3.Count = 10 then
   	P_Tem3.Count := 0;
   	P_Tem3.MeanStart := 1;
   end_if;
   P_Tem3.CurrentValue := Local:3:I.Ch06.Data;
   if P_Tem3.MeanStart then
   	P_Tem3.Mean10 := (P_Tem3.PreviousValue0 + P_Tem3.PreviousValue1 + P_Tem3.PreviousValue2 + P_Tem3.PreviousValue3 + P_Tem3.PreviousValue4 + P_Tem3.PreviousValue5 + P_Tem3.PreviousValue6 + P_Tem3.PreviousValue7 + P_Tem3.PreviousValue8 + P_Tem3.PreviousValue9)/10;
   	P_Tem3.StanDev := SQRT(((P_Tem3.PreviousValue0 - P_Tem3.Mean10)**2 + (P_Tem3.PreviousValue1 - P_Tem3.Mean10)**2 + (P_Tem3.PreviousValue2 - P_Tem3.Mean10)**2 + (P_Tem3.PreviousValue3 - P_Tem3.Mean10)**2 + (P_Tem3.PreviousValue4 - P_Tem3.Mean10)**2 + (P_Tem3.PreviousValue5 - P_Tem3.Mean10)**2 + (P_Tem3.PreviousValue6 - P_Tem3.Mean10)**2 + (P_Tem3.PreviousValue7 - P_Tem3.Mean10)**2 + (P_Tem3.PreviousValue8 - P_Tem3.Mean10)**2 + (P_Tem3.PreviousValue9 - P_Tem3.Mean10)**2)/10);
   end_if;
END_ROUTINE

ROUTINE Update_P_Tem4   (* structured text *)
   case P_Tem4.Count of
   	0: P_Tem4.PreviousValue0 := P_Tem4.CurrentValue;
   	1: P_Tem4.PreviousValue1 := P_Tem4.CurrentValue;
   	2: P_Tem4.PreviousValue2 := P_Tem4.CurrentValue;
   	3: P_Tem4.PreviousValue3 := P_Tem4.CurrentValue;
   	4: P_Tem4.PreviousValue4 := P_Tem4.CurrentValue;
   	5: P_Tem4.PreviousValue5 := P_Tem4.CurrentValue;
   	6: P_Tem4.PreviousValue6 := P_Tem4.CurrentValue;
   	7: P_Tem4.PreviousValue7 := P_Tem4.CurrentValue;
   	8: P_Tem4.PreviousValue8 := P_Tem4.CurrentValue;
   	9: P_Tem4.PreviousValue9 := P_Tem4.CurrentValue;
   end_case;
   P_Tem4.Count := P_Tem4.Count + 1;
   if P_Tem4.Count = 10 then
   	P_Tem4.Count := 0;
   	P_Tem4.MeanStart := 1;
   end_if;
   P_Tem4.CurrentValue := Local:3:I.Ch07.Data;
   if P_Tem4.MeanStart then
   	P_Tem4.Mean10 := (P_Tem4.PreviousValue0 + P_Tem4.PreviousValue1 + P_Tem4.PreviousValue2 + P_Tem4.PreviousValue3 + P_Tem4.PreviousValue4 + P_Tem4.PreviousValue5 + P_Tem4.PreviousValue6 + P_Tem4.PreviousValue7 + P_Tem4.PreviousValue8 + P_Tem4.PreviousValue9)/10;
   	P_Tem4.StanDev := SQRT(((P_Tem4.PreviousValue0 - P_Tem4.Mean10)**2 + (P_Tem4.PreviousValue1 - P_Tem4.Mean10)**2 + (P_Tem4.PreviousValue2 - P_Tem4.Mean10)**2 + (P_Tem4.PreviousValue3 - P_Tem4.Mean10)**2 + (P_Tem4.PreviousValue4 - P_Tem4.Mean10)**2 + (P_Tem4.PreviousValue5 - P_Tem4.Mean10)**2 + (P_Tem4.PreviousValue6 - P_Tem4.Mean10)**2 + (P_Tem4.PreviousValue7 - P_Tem4.Mean10)**2 + (P_Tem4.PreviousValue8 - P_Tem4.Mean10)**2 + (P_Tem4.PreviousValue9 - P_Tem4.Mean10)**2)/10);
   end_if;
END_ROUTINE
END_PROGRAM

PROGRAM SafetyProgram   (* main routine MainRoutine, safety *)
VAR
   B_Stage1 : BOOL;
   B_Stage2 : BOOL;
END_VAR

ROUTINE Eval_Bat   (* ladder *)
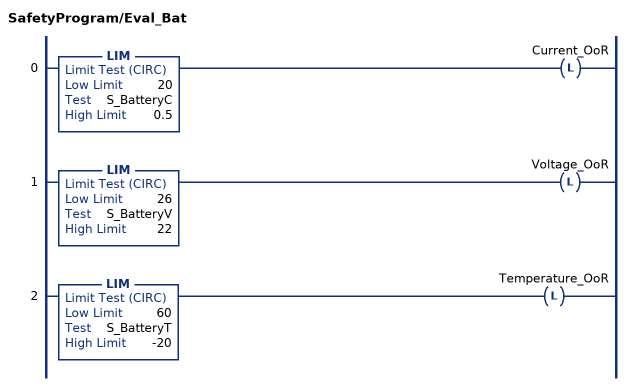
   0: LIM(20,S_BatteryC,0.5)OTL(Current_OoR);
   1: LIM(26,S_BatteryV,22)OTL(Voltage_OoR);
   2: LIM(60,S_BatteryT,-20)OTL(Temperature_OoR);
END_ROUTINE

ROUTINE Eval_Brake   (* ladder *)
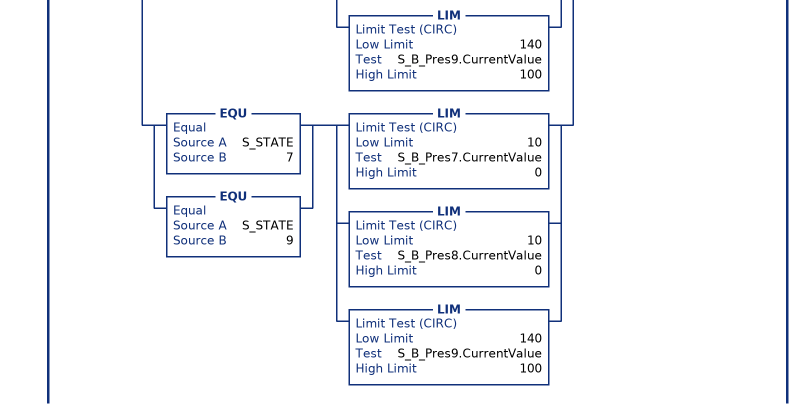
   0: [OTL(B_Stage1) [[LIM(105,S_B_Pres0.CurrentValue,95) ,LIM(105,S_B_Pres1.CurrentValue,95) ,LIM(30,S_B_Tem0.CurrentValue,20) ] ,[LIM(1,S_STATE,5) ,EQU(S_STATE,8) ] [LIM(16,S_B_Pres2.CurrentValue,12) ,LIM(16,S_B_Pres3.CurrentValue,12) ,LIM(170,S_B_Pres4.CurrentValue,150) ] ,[EQU(S_STATE,6) ,EQU(S_STATE,10) ] [LIM(105,S_B_Pres2.CurrentValue,95) ,LIM(105,S_B_Pres3.CurrentValue,95) ,LIM(140,S_B_Pres4.CurrentValue,100) ] ,[EQU(S_STATE,7) ,EQU(S_STATE,9) ] [LIM(10,S_B_Pres2.CurrentValue,0) ,LIM(10,S_B_Pres3.CurrentValue,0) ,LIM(140,S_B_Pres4.CurrentValue,100) ] ] MOV(1,S_Brake_Sub1) ,OTL(B_Stage2) [[LIM(105,S_B_Pres5.CurrentValue,95) ,LIM(105,S_B_Pres6.CurrentValue,95) ,LIM(30,S_B_Tem1.CurrentValue,20) ] ,[LIM(1,S_STATE,5) ,EQU(S_STATE,8) ] [LIM(16,S_B_Pres7.CurrentValue,12) ,LIM(16,S_B_Pres8.CurrentValue,12) ,LIM(170,S_B_Pres9.CurrentValue,150) ] ,[EQU(S_STATE,6) ,EQU(S_STATE,10) ] [LIM(105,S_B_Pres7.CurrentValue,95) ,LIM(105,S_B_Pres8.CurrentValue,95) ,LIM(140,S_B_Pres9.CurrentValue,100) ] ,[EQU(S_STATE,7) ,EQU(S_STATE,9) ] [LIM(10,S_B_Pres7.CurrentValue,0) ,LIM(10,S_B_Pres8.CurrentValue,0) ,LIM(140,S_B_Pres9.CurrentValue,100) ] ] MOV(1,S_Brake_Sub2) ];
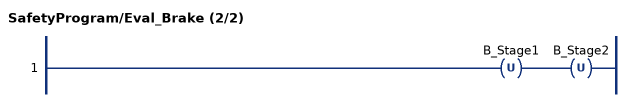
   1: OTU(B_Stage1)OTU(B_Stage2);
END_ROUTINE

ROUTINE Eval_Comm   (* ladder *)
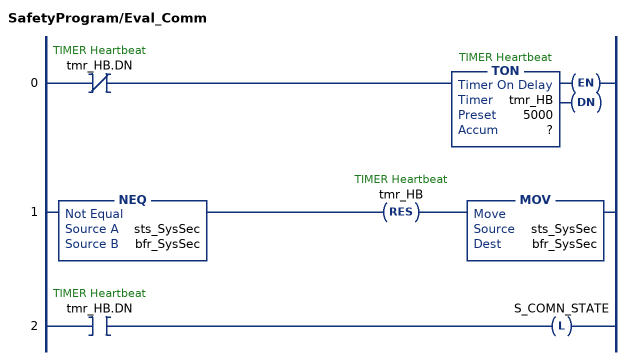
   0: XIO(tmr_HB.DN)TON(tmr_HB,?,?);
   1: NEQ(sts_SysSec,bfr_SysSec)RES(tmr_HB)MOV(sts_SysSec,bfr_SysSec);
   2: XIC(tmr_HB.DN)OTL(S_COMN_STATE);
END_ROUTINE

ROUTINE Eval_Prop   (* ladder *)
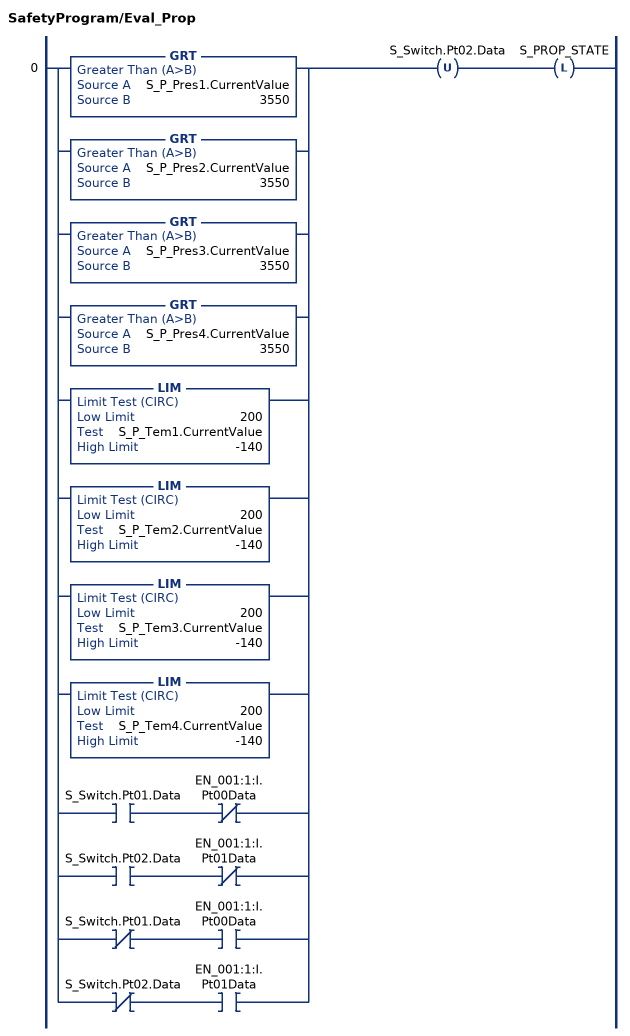
   0: [GRT(S_P_Pres1.CurrentValue,3550) ,GRT(S_P_Pres2.CurrentValue,3550) ,GRT(S_P_Pres3.CurrentValue,3550) ,GRT(S_P_Pres4.CurrentValue,3550) ,LIM(200,S_P_Tem1.CurrentValue,-140) ,LIM(200,S_P_Tem2.CurrentValue,-140) ,LIM(200,S_P_Tem3.CurrentValue,-140) ,LIM(200,S_P_Tem4.CurrentValue,-140) ,XIC(S_Switch.Pt01.Data) XIO(EN_001:1:I.Pt00Data) ,XIC(S_Switch.Pt02.Data) XIO(EN_001:1:I.Pt01Data) ,XIO(S_Switch.Pt01.Data) XIC(EN_001:1:I.Pt00Data) ,XIO(S_Switch.Pt02.Data) XIC(EN_001:1:I.Pt01Data) ]OTU(S_Switch.Pt02.Data)OTL(S_PROP_STATE);
END_ROUTINE

ROUTINE MainRoutine   (* ladder *)
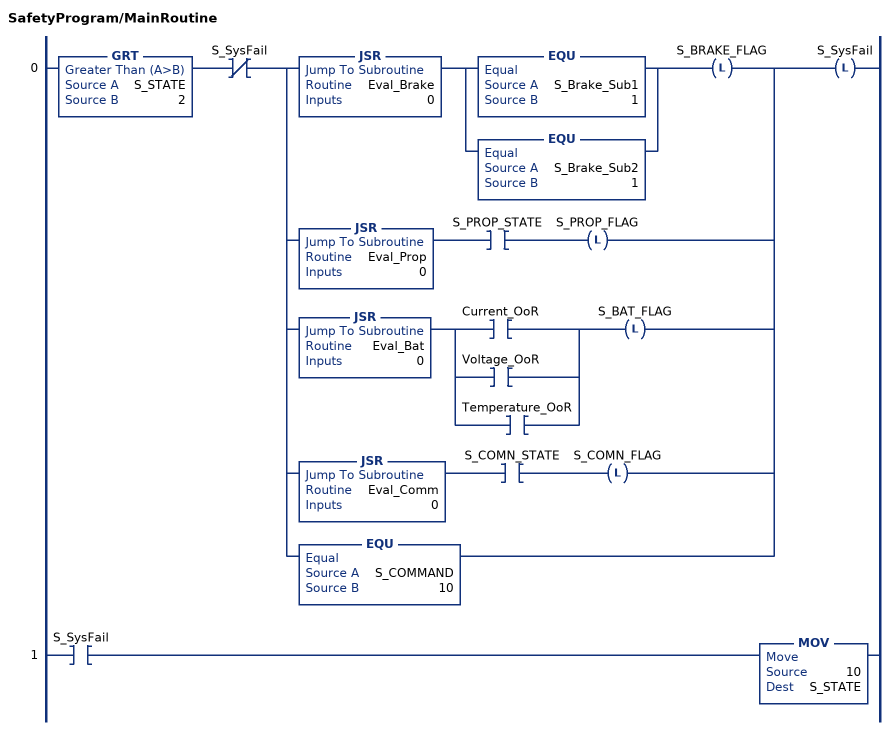
   0: GRT(S_STATE,2)XIO(S_SysFail)[JSR(Eval_Brake,0) [EQU(S_Brake_Sub1,1) ,EQU(S_Brake_Sub2,1) ] OTL(S_BRAKE_FLAG) ,JSR(Eval_Prop,0) XIC(S_PROP_STATE) OTL(S_PROP_FLAG) ,JSR(Eval_Bat,0) [XIC(Current_OoR) ,XIC(Voltage_OoR) ,XIC(Temperature_OoR) ] OTL(S_BAT_FLAG) ,JSR(Eval_Comm,0) XIC(S_COMN_STATE) OTL(S_COMN_FLAG) ,EQU(S_COMMAND,10) ]OTL(S_SysFail);
   1: XIC(S_SysFail)MOV(10,S_STATE);
END_ROUTINE
END_PROGRAM
